TYPE "FeedMachine_DataOut"
VERSION : 0.1
// Block: FeedMachine_DataOut
   STRUCT
      Fan_M_Contactor : Bool;
   END_STRUCT;

END_TYPE
